Universal Robots PolyScope program: orange_Museum.urp

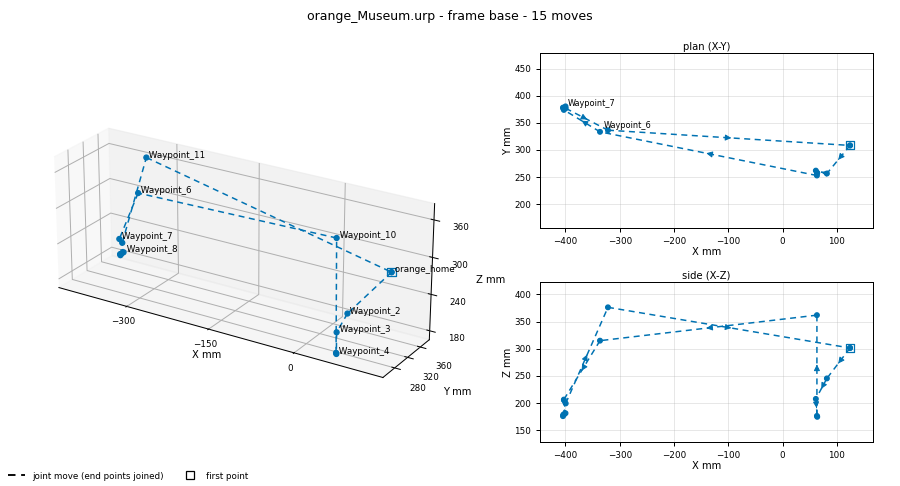
[picture p0: tool path of orange_Museum.urp in frame base, 15 of 15 moves have a stored position in this frame; points joined in program order, loops and branches not executed]
Program orange_Museum (installation=default directory=/programs/usbdisk/Zahra1/orangi createdIn=5.11.11.1010533 lastSavedIn=5.11.11.1010533 robotSerialNumber=20205300864)
Calibrated DH parameters: a=[-0.000166, -0.243494, -0.153108, 0.000057, -0.000123, 0]; d=[0.151897, -1.34267, 53.988124, -52.514559, 0.085283, 0.092193]; alpha=[1.572472, -0.003756, 0.002824, 1.570807, -1.572621, 0]; deltaTheta=[0, 0.020704, 7.033215, -0.770746, 0.000004, 0]
Robot Program (runOnlyOnce=true)
  MoveJ speed 60 deg/s, acceleration 80 deg/s^2 (useActiveTCP=true) feature=Base
    Waypoint orange_home: TCP in base x=124.286 y=308.277 z=301.462 mm, rx=2.2499 ry=-2.1846 rz=-0.0963 rad; joints [-269.66, -91.226, -90.279, -86.086, 92.69, 808.818] deg
    URCap Gripper (Robotiq_Grippers, Robotiq Inc.) dataModel(position=32.15686274509804, force=50.0, speed=18.0, positionInDouble=32.15686274509804, forceInDouble=50.0, speedInDouble=18.0, slaveIds=[9], blocking=true, robotCompliant=false)
    Waypoint Waypoint_2: TCP in base x=81.625 y=256.499 z=245.371 mm, rx=-3.1021 ry=0.0993 rz=0.1401 rad; joints [-260.494, -76.625, -118.753, -71.532, 94.768, 733.439] deg
    Waypoint Waypoint_3: TCP in base x=61.297 y=261.858 z=207.616 mm, rx=-3.1329 ry=0.0132 rz=0.0097 rad; joints [-254.265, -79.826, -126.04, -63.454, 90.302, 736.379] deg
    Waypoint Waypoint_4: TCP in base x=63.874 y=257.722 z=174.628 mm, rx=-3.1157 ry=0.0576 rz=-0.0097 rad; joints [-254.227, -83.738, -133.629, -51.246, 89.325, 738.077] deg
    URCap Gripper (Robotiq_Grippers, Robotiq Inc.) dataModel(position=83.15686274509804, force=73.0, speed=18.0, positionInDouble=83.15686274509804, forceInDouble=73.0, speedInDouble=18.0, slaveIds=[9], blocking=true, robotCompliant=false)
    Waypoint Waypoint_5: motionParameters(jointSpeed=0.698132 jointAcceleration=0.349066 cartesianSpeed=0.25 cartesianAcceleration=1.2); TCP in base x=63.282 y=257.862 z=176.274 mm, rx=-3.1141 ry=0.0575 rz=0.0008 rad; joints [-254.232, -83.474, -133.4, -51.535, 89.671, 738.072] deg
    Waypoint Waypoint_10: TCP in base x=63.267 y=252.883 z=361.941 mm, rx=-3.1142 ry=0.0574 rz=0.0007 rad; joints [-253.809, -74.367, -87.857, -106.192, 89.609, 738.362] deg
    Waypoint Waypoint_6: TCP in base x=-336.397 y=333.329 z=314.919 mm, rx=-0.0274 ry=-3.049 rz=-0.0384 rad; joints [-208.941, -130.451, -32.753, -101.355, 91.09, 602.162] deg
    Waypoint Waypoint_7: TCP in base x=-402.964 y=373.738 z=206.361 mm, rx=0.0203 ry=-2.9288 rz=-0.0698 rad; joints [-209.692, -155.213, -18.049, -84.751, 93.528, 599.837] deg
    Waypoint Waypoint_8: TCP in base x=-399.927 y=380.221 z=181.259 mm, rx=-0.0612 ry=-2.9325 rz=0.02 rad; joints [-210.946, -158.065, -18.189, -83.625, 96.39, 601.966] deg
    Waypoint Waypoint_12: TCP in base x=-402.265 y=377.83 z=179.256 mm, rx=-0.0433 ry=-2.9512 rz=-0.0014 rad; joints [-210.385, -158.187, -18.187, -83.999, 95.122, 601.682] deg
    Waypoint Waypoint_9: motionParameters(jointSpeed=0.698132 jointAcceleration=0.174533 cartesianSpeed=0.25 cartesianAcceleration=1.2); TCP in base x=-403.871 y=376.159 z=178.6 mm, rx=-0.036 ry=-2.9626 rz=-0.0154 rad; joints [-210.004, -158.255, -18.06, -84.343, 94.297, 601.693] deg
    Waypoint Waypoint_1: TCP in base x=-404.609 y=377.966 z=175.858 mm, rx=-0.0399 ry=-2.9637 rz=-0.0076 rad; joints [-210.168, -159.912, -15.278, -85.68, 94.539, 601.682] deg
    URCap Gripper (Robotiq_Grippers, Robotiq Inc.) dataModel(position=56.07843137254902, force=8.0, speed=2.0, positionInDouble=56.07843137254902, forceInDouble=8.0, speedInDouble=2.0, slaveIds=[9], blocking=true, robotCompliant=false)
    Waypoint Waypoint_13: TCP in base x=-399.532 y=376.683 z=199.31 mm, rx=-0.0428 ry=-2.9529 rz=-0.0176 rad; joints [-210.315, -157.024, -15.252, -87.873, 94.515, 601.685] deg
    Waypoint Waypoint_11: TCP in base x=-321.712 y=336.341 z=376.361 mm, rx=-0.0968 ry=-2.9018 rz=-0.1122 rad; joints [-210.421, -130.999, -18.094, -106.805, 92.37, 603.68] deg
    Waypoint orange_home: TCP in base x=124.286 y=308.277 z=301.462 mm, rx=2.2499 ry=-2.1846 rz=-0.0963 rad; joints [-269.66, -91.226, -90.279, -86.086, 92.69, 808.818] deg
